FUNCTION_BLOCK E_CTUD (* Event-Driven Up/Down Counter *)
  (* Standard: 61499-1-A; Classification: Event-driven blocks; Function: Up/Down counter *)
  (* Version 0.0, 2006-09-07, JHC, Holobloc Inc *)
  (* Compiler header: package fb.rt.events; *)
  (* Compiler Java Sun JDK 1.5.0 *)
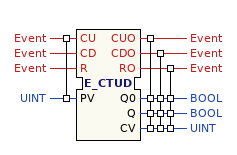
  EVENT_INPUT
    CU WITH PV; (* Count Up *)
    CD; (* Count Down *)
    R; (* Reset *)
  END_EVENT
  EVENT_OUTPUT
    CUO WITH Q, CV, Q0; (* Count Up Output Event *)
    CDO WITH Q, CV, Q0; (* Count Down Output Event *)
    RO WITH Q, CV, Q0; (* Reset Output Event *)
  END_EVENT
  VAR_INPUT
    PV : UINT; (* Preset Value *)
  END_VAR
  VAR_OUTPUT
    Q0 : BOOL; (* CV==0 *)
    Q : BOOL; (* CV>=PV *)
    CV : UINT;
  END_VAR
END_FUNCTION_BLOCK
